# EPICS autosave request: ipApp/Db/Oxford_CS800_status.req
$(P)$(R)status_packet.SCAN
$(P)$(R)status_packet.TMOD
$(P)$(R)status_packet.OEOS
$(P)$(R)status_packet.IEOS
$(P)$(R)status_packet.OFMT
$(P)$(R)status_packet.IFMT
$(P)$(R)status_packet.TMOT
$(P)$(R)status_packet.NRRD
